FUNCTION_BLOCK FB_Barn EXTENDS FB_Station
VAR
END_VAR

METHOD AutoImport : PVOID
VAR_INPUT
	Egg			: INT;
	Chicken		: INT;
END_VAR
VAR
	stTempEgg			: ST_Unit;
	iTempEgg			: INT;
	stTempChicken		: ST_Unit;
	iTempChicken		: INT;
END_VAR
FOR iTempEgg := 1 TO Egg BY 1 DO
	stTempEgg.eType := 0;
	stTempEgg.iHitPoint := 30;
	stTempEgg.iProgress := 0;
	UnitImport(stTempEgg);
END_FOR

FOR iTempChicken := 1 TO Chicken BY 1 DO
	stTempChicken.eType := 1;
	stTempChicken.iHitPoint := 30;
	stTempChicken.iProgress := 0;
	UnitImport(stTempChicken);
END_FOR
END_METHOD

METHOD Run : BOOL
VAR_INPUT
END_VAR
iMaxUnit := iCurLevel * 20;
END_METHOD

END_FUNCTION_BLOCK

(* stored: Version 1.1.0.1, ProductVersion 3.1.4024.12
   POU FB_Barn: Id {cf9725ae-d3e0-4439-8c00-4d7018d0d139}, SpecialFunc None
   Method AutoImport: Id {efad2820-81ad-4919-9d7c-23f161d21edd}
   Method Run: Id {933056ec-e406-414c-8d4f-50f2eea35eb3} *)
